TYPE E_FFMode :
(
    FF    := 0,    // Standard FF
    KvFF  := 1     // Kv-based FF with polynomial for spool
);
END_TYPE

(* stored: Version 1.1.0.1
   DUT E_FFMode: Id {b863c1e8-012e-42a0-b36f-00427d6c0534} *)
